FUNCTION_BLOCK FB_Power
VAR_INPUT
	bEnable			: BOOL := FALSE;
	fOverride		: LREAL := 1.0;
END_VAR
VAR_IN_OUT
	stAxisAcs		: ARRAY[1..4] OF AXIS_REF;
	stAxisMcs		: ARRAY[1..3] OF AXIS_REF;
END_VAR
VAR_OUTPUT
	bAllAxesReady	: BOOL := FALSE;
	bError			: BOOL;
END_VAR
VAR
	fbPowerAcs		: ARRAY [1..4] OF MC_Power;
	fbPowerMcs	 	: ARRAY [1..3] OF MC_Power;
	i				: UINT;
END_VAR

bAllAxesReady := TRUE;
bError := FALSE;

FOR i:=1 TO 4 DO
	fbPowerAcs[i](Axis:=stAxisAcs[i],
		Enable			:= bEnable,
		Enable_Positive	:= bEnable,
		Enable_Negative	:= bEnable
	);
	
	IF i <= 3 THEN
		fbPowerMcs[i](Axis:=stAxisMcs[i],
			Enable			:= bEnable,
			Enable_Positive	:= bEnable,
			Enable_Negative	:= bEnable
		);
		
		bAllAxesReady := bAllAxesReady AND fbPowerAcs[i].Status AND fbPowerMcs[i].Status; 
		bError := bError OR fbPowerAcs[i].Error OR fbPowerMcs[i].Error;
		
	ELSE
		bAllAxesReady := bAllAxesReady AND fbPowerAcs[i].Status;
		bError := bError OR fbPowerAcs[i].Error;
	END_IF
	 
END_FOR

END_FUNCTION_BLOCK

(* stored: Version 1.1.0.1, ProductVersion 3.1.4024.5
   POU FB_Power: Id {f4074599-01e5-40b3-b609-a36846c6bc1f}, SpecialFunc None *)
